(*
SPDX-FileCopyrightText: © 2026 Oleksandr Tiutyk <trofimich@gmail.com>
SPDX-License-Identifier: MIT
License: https://opensource.org/license/mit
*)

(*!
<summary>Reports an operation that requires an element in an empty collection.</summary>
<description>
The caller detects the condition; this exception does not inspect or modify the collection or destination.
Uses the GeneralException task-local cycle lifetime and throw rules. Dynamic copies are explicitly registered
by Clone after construction; plain __NEW does not transfer ownership to the task manager.
</description>
*)

{attribute 'enable_dynamic_creation'}
{attribute 'no_explicit_call' := 'do not call this function block directly'}
FUNCTION_BLOCK CollectionEmptyException EXTENDS GeneralException IMPLEMENTS ICollectionEmptyException
VAR_STAT
	//! <summary>Class name shared by all instances of this function block.</summary>
	{attribute 'hide'} 
	_ClassName : STRING := __POUNAME();
END_VAR

{attribute 'monitoring' := 'call'}
PROPERTY ClassName : REFERENCE TO STRING
GET
ClassName REF= _ClassName;
END_GET
END_PROPERTY

(*!
<summary>Creates a clone of this concrete exception type.</summary>
<description>
Copies GeneralException fields and timestamps. The clone belongs to DynamicMemoryManager until cleanup of the
creating task; callers must not delete it. Allocation failure is terminal. Registers the newly constructed
instance before copying payload, outside FB_init. Registration failure releases the unregistered instance and
raises a terminal error; copy failure leaves the registered instance owned by the task manager for cleanup.
Custom overrides must follow the same ownership sequence.
</description>
*)
METHOD Clone : IObject
VAR
	exceptionClone : POINTER TO CollectionEmptyException;
END_VAR
exceptionClone := __NEW(CollectionEmptyException);

IF exceptionClone = 0 THEN
	DynamicMemoryManager.RaiseAllocationFailure();
END_IF

DynamicMemoryManager.RegisterAutoDisposedObject(autoDisposedObject := exceptionClone^);

exceptionClone^.CopyGeneralFields(sourceException := THIS^);

Clone := exceptionClone^;
END_METHOD

(*!
<summary>Provides the library namespace used in diagnostics.</summary>
<description>
Borrowed read-only reference to the compiler-initialized library namespace; no ownership transfer.
</description>
*)
{attribute 'monitoring' := 'call'}
PROPERTY NamespaceName : REFERENCE TO STRING
GET
NamespaceName REF= CurrentNamespace.Name;
END_GET
END_PROPERTY

(*!
<summary>Reports the byte size of this concrete instance.</summary>
<description>
Uses XSIZEOF on the instance. Does not include separately allocated payloads or prove that an arbitrary
address is valid.
</description>
*)
{attribute 'monitoring' := 'call'}
PROPERTY SelfSize : ULINT
GET
SelfSize := XSIZEOF(THIS^);
END_GET
END_PROPERTY

(*!
<summary>Builds the diagnostic and raises this exception through GeneralException.</summary>
<description>
Copies the supplied diagnostic data, sets error code to zero and supplies no inner exception. Call only in a
cyclic task, not during FB_init. The caller must already have detected the reported condition.
</description>
<param name="collectionName">Collection name used in the diagnostic.</param>
*)
METHOD Throw
VAR_INPUT
	sourceNamespaceName : STRING;
	sourceClassName : STRING;
	sourcePOUName : STRING;
	sourcePosition : STRING;
	collectionName : WSTRING;
END_VAR
VAR
	message : ERROR_MESSAGE;
END_VAR
message := WideStrings.Concat255("Collection '", collectionName, "' is empty");

InternalThrow(
	sourceNamespaceName := sourceNamespaceName,
	sourceClassName := sourceClassName,
	sourcePOUName := sourcePOUName,
	sourcePosition := sourcePosition,
	message := message,
	errorCode := 0,
	innerException := 0
);
END_METHOD

END_FUNCTION_BLOCK

(* stored: Version 1.1.0.1
   POU CollectionEmptyException: Id {4bed74e9-976c-48cb-976a-f2975ddf9c18}, SpecialFunc None
   Property ClassName: Id {abd18078-730a-4c0b-a477-d30a629c8651}
   Get Get: Id {80f03232-533a-4819-aab5-ef22ad3012ae}
   Method Clone: Id {00a28a02-e5ef-4b60-8d41-fed22a2a3cf3}
   Property NamespaceName: Id {5cd7d887-5c22-49ba-b54a-d3b90c5987b2}
   Get Get: Id {a7028650-cd01-4152-9dbe-c33d8b203ef3}
   Property SelfSize: Id {f5526be1-75ca-421e-a992-13ae56664348}
   Get Get: Id {0285d1b7-0819-420f-b62e-f5826833bfbb}
   Method Throw: Id {a609eb33-c8ea-4f01-9d83-0cf925cf5871} *)
